RoboDK station: kr30 cnc template amana 46348 - paulina NEW THING.rdk

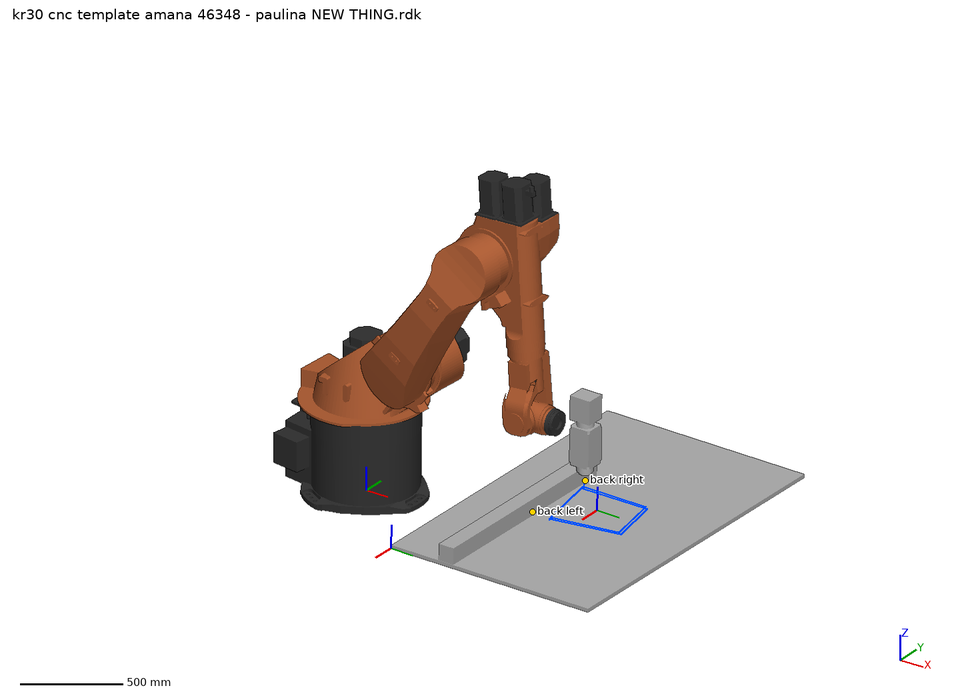
[picture v0: the station drawn from its stored meshes, robots at their saved joint values, targets as dots, program paths as lines]
Station kr30 cnc template amana 46348 - paulina NEW THING. Poses are relative to the parent item; angles as X-Y-Z fixed-axis rotations.
  - frame KUKA KR 30 HA Base at (0, 0, 0) mm
    - robot KUKA KR 30 HA: 6 axes, payload 30 kg, reach 2033 mm, repeatability 0.05 mm, weight 665 kg
        modified DH rows (alpha deg, a mm, theta deg, d mm): 0, 0, 0, 815; -90, 350, 0, 0; 0, 850, -90, 0; -90, 145, 0, 820; 90, 0, 0, 0; -90, 0, 180, 170
        joint limits [-185, -135, -120, -350, -119, -350] to [185, 35, 158, 350, 119, 350]; home [0, -90, 90, 0, 0, 0]; saved at [3.324, -56.878, 143.017, 183.529, 85.332, -180.023]
      - tool rc90 spindle mm, TCP at (267.95, 0.68, 160.99) mm, size 110 x 421.3 x 118 mm, geometry from rc90 spindle mm.stl
    - frame Tabletop at (921.82, -1104.91, 385) mm, rotated rx -0.93 ry -0.21 rz -89.9 deg
      - object tabletop CHECK HEIGHT at (-1839.9, 0, 0) mm, size 1839.9 x 1168.4 x 19 mm, geometry from kr30 tabletop mm.stl
      - object kr30 pipe jig base at (-1220, -610.6, 0) mm, size 1217.6 x 88.9 x 88.9 mm, geometry from kr30 pipe jig base.stl
      - frame Frame 3 at (-850, 630, 55.44) mm
      - target back right (Cartesian target) at (-1090.62, 392.95, 52.9) mm, rotated rx -9.38 ry 89.87 rz 80.74 deg; joints [0.828, -55.747, 144.821, 181.035, 88.274, -179.786] of KUKA KR 30 HA
      - target back left (Cartesian target) at (-646.79, 387.88, 55.43) mm, rotated rx -9.38 ry 89.87 rz 80.73 deg; joints [25.002, -54.059, 137.701, 205.384, 83.45, -182.49] of KUKA KR 30 HA
  - machining project Machining Settings: C:/Users/Research Office/Downloads/C1.apt | rotZ(0) | rotX(0)*rotY(0) | onStart | onPathStart | onApproach | onPoint | onRetract | onFinish | SetTool(%1) | onPathFinish
  - program Machining (400 instructions, listed below)
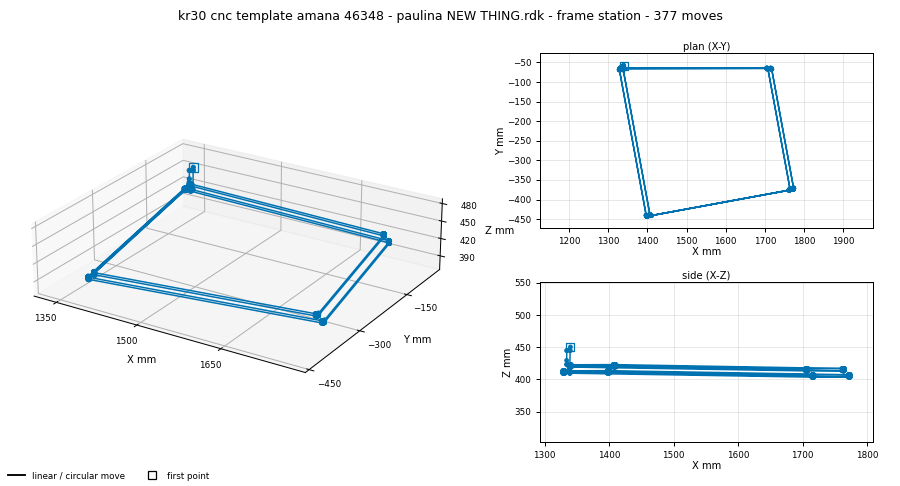
[picture p0: tool path of kr30 cnc template amana 46348 - paulina NEW THING.rdk in frame station, 377 of 377 moves have a stored position in this frame; points joined in program order, loops and branches not executed]

--- program Machining (robot KUKA KR 30 HA) ---
  Smooth(10)
  Print: /'1001'
  Print: /''
  Print: /'90 deg cut'
  Call SetTool(2)
  Set speed (100.0 mm/s)
  Set Ref.: Frame 3
  Set Tool: rc90 spindle mm
  Show rc90 spindle mm
  MoveJ 1 to (-195.95, -211.4, 20.67) mm, rotated rx -2.36 ry 89.88 rz 87.74 deg; joints [3.323, -57.284, 143.059, 183.53, 84.969, -180.046]
  MoveL 2 to (-192.49, -216.97, 15) mm, rotated rx 0 ry 90 rz 90.11 deg; joints [3.542, -56.953, 143.366, -176.241, 85.489, 179.974]
  MoveL 3 to (-192.49, -216.97, 15) mm, rotated rx 0 ry 90 rz 90.11 deg; joints [3.542, -56.953, 143.366, -176.241, 85.489, 179.974]
  Set speed (100.0 mm/s)
  MoveL 4 to (-192.49, -216.97, -0.32) mm, rotated rx 0 ry 90 rz 90.11 deg; joints [3.546, -55.577, 143.206, -176.242, 86.702, 180.054]
  Set speed (25.4 mm/s)
  MoveL 5 to (-192.49, -216.97, -6.37) mm, rotated rx 0 ry 90 rz 90.11 deg; joints [3.548, -55.032, 143.136, -176.242, 87.175, 180.085]
  MoveL 6 to (-192.02, -216.54, -7) mm, rotated rx 0 ry 90 rz 90.11 deg; joints [3.573, -54.966, 143.095, -176.217, 87.201, 180.086]
  Set speed (38.1 mm/s)
  MoveL 7 to (-187.83, -212.73, -7) mm, rotated rx 0 ry 90 rz 90.11 deg; joints [3.796, -54.884, 142.796, -175.994, 86.985, 180.063]
  MoveL 8 to (-187.84, -211.79, -7) mm, rotated rx 0 ry 90 rz 90.11 deg; joints [3.792, -54.864, 142.727, -175.997, 86.935, 180.06]
  Set speed (76.2 mm/s)
  MoveL 9 to (-188.01, -211.61, -7) mm, rotated rx 0 ry 90 rz 90.11 deg; joints [3.782, -54.861, 142.715, -176.007, 86.927, 180.06]
  MoveL 10 to (-188.15, -211.43, -7) mm, rotated rx 0 ry 90 rz 90.11 deg; joints [3.773, -54.857, 142.703, -176.016, 86.918, 180.06]
  MoveL 11 to (-188.32, -211.19, -7) mm, rotated rx 0 ry 90 rz 90.11 deg; joints [3.762, -54.852, 142.686, -176.027, 86.906, 180.059]
  MoveL 12 to (-188.46, -210.95, -7) mm, rotated rx 0 ry 90 rz 90.11 deg; joints [3.754, -54.848, 142.669, -176.035, 86.894, 180.059]
  MoveL 13 to (-188.57, -210.71, -7) mm, rotated rx 0 ry 90 rz 90.11 deg; joints [3.746, -54.843, 142.652, -176.042, 86.882, 180.058]
  MoveL 14 to (-188.66, -210.47, -7) mm, rotated rx 0 ry 90 rz 90.11 deg; joints [3.741, -54.838, 142.634, -176.048, 86.869, 180.057]
  MoveL 15 to (-188.72, -210.23, -7) mm, rotated rx 0 ry 90 rz 90.11 deg; joints [3.736, -54.833, 142.617, -176.053, 86.857, 180.057]
  MoveL 16 to (-188.77, -209.99, -7) mm, rotated rx 0 ry 90 rz 90.11 deg; joints [3.732, -54.828, 142.6, -176.056, 86.845, 180.056]
  MoveL 17 to (-188.8, -209.74, -7) mm, rotated rx 0 ry 90 rz 90.11 deg; joints [3.73, -54.823, 142.582, -176.059, 86.832, 180.055]
  MoveL 18 to (-188.81, -209.5, -7) mm, rotated rx 0 ry 90 rz 90.11 deg; joints [3.728, -54.818, 142.564, -176.06, 86.82, 180.054]
  MoveL 19 to (-188.81, 153.51, -7) mm, rotated rx 0 ry 90 rz 90.11 deg; joints [2.724, -44.301, 113.966, -176.857, 68.761, 179.117]
  MoveL 20 to (-188.81, 153.99, -7) mm, rotated rx 0 ry 90 rz 90.11 deg; joints [2.723, -44.283, 113.924, -176.858, 68.736, 179.116]
  MoveL 21 to (-188.8, 154.23, -7) mm, rotated rx 0 ry 90 rz 90.11 deg; joints [2.723, -44.275, 113.904, -176.858, 68.724, 179.116]
  MoveL 22 to (-188.76, 154.47, -7) mm, rotated rx 0 ry 90 rz 90.11 deg; joints [2.724, -44.266, 113.883, -176.856, 68.712, 179.115]
  MoveL 23 to (-188.71, 154.71, -7) mm, rotated rx 0 ry 90 rz 90.11 deg; joints [2.725, -44.257, 113.862, -176.854, 68.7, 179.113]
  MoveL 24 to (-188.64, 154.96, -7) mm, rotated rx 0 ry 90 rz 90.11 deg; joints [2.728, -44.248, 113.841, -176.851, 68.688, 179.112]
  MoveL 25 to (-188.55, 155.2, -7) mm, rotated rx 0 ry 90 rz 90.11 deg; joints [2.731, -44.24, 113.82, -176.848, 68.676, 179.11]
  MoveL 26 to (-188.43, 155.44, -7) mm, rotated rx 0 ry 90 rz 90.11 deg; joints [2.735, -44.231, 113.798, -176.843, 68.664, 179.107]
  MoveL 27 to (-188.35, 155.57, -7) mm, rotated rx 0 ry 90 rz 90.11 deg; joints [2.738, -44.226, 113.787, -176.839, 68.657, 179.106]
  MoveL 28 to (-188.27, 155.7, -7) mm, rotated rx 0 ry 90 rz 90.11 deg; joints [2.741, -44.221, 113.775, -176.836, 68.65, 179.104]
  MoveL 29 to (-188.18, 155.83, -7) mm, rotated rx 0 ry 90 rz 90.11 deg; joints [2.745, -44.216, 113.763, -176.832, 68.644, 179.103]
  MoveL 30 to (-188.08, 155.96, -7) mm, rotated rx 0 ry 90 rz 90.11 deg; joints [2.749, -44.211, 113.752, -176.827, 68.637, 179.101]
  MoveL 31 to (-187.95, 156.11, -7) mm, rotated rx 0 ry 90 rz 90.11 deg; joints [2.754, -44.206, 113.739, -176.822, 68.629, 179.098]
  MoveL 32 to (-187.8, 156.26, -7) mm, rotated rx 0 ry 90 rz 90.11 deg; joints [2.76, -44.2, 113.725, -176.815, 68.622, 179.096]
  MoveL 33 to (-187.66, 156.38, -7) mm, rotated rx 0 ry 90 rz 90.11 deg; joints [2.765, -44.195, 113.714, -176.809, 68.615, 179.093]
  MoveL 34 to (-187.52, 156.49, -7) mm, rotated rx 0 ry 90 rz 90.11 deg; joints [2.771, -44.191, 113.704, -176.803, 68.61, 179.091]
  MoveL 35 to (-187.28, 156.65, -7) mm, rotated rx 0 ry 90 rz 90.11 deg; joints [2.781, -44.185, 113.689, -176.793, 68.601, 179.087]
  MoveL 36 to (-187.04, 156.78, -7) mm, rotated rx 0 ry 90 rz 90.11 deg; joints [2.79, -44.18, 113.677, -176.782, 68.594, 179.082]
  MoveL 37 to (-186.8, 156.89, -7) mm, rotated rx 0 ry 90 rz 90.11 deg; joints [2.8, -44.176, 113.667, -176.772, 68.588, 179.078]
  MoveL 38 to (-186.55, 156.97, -7) mm, rotated rx 0 ry 90 rz 90.11 deg; joints [2.81, -44.172, 113.658, -176.761, 68.584, 179.074]
  MoveL 39 to (-186.31, 157.03, -7) mm, rotated rx 0 ry 90 rz 90.11 deg; joints [2.82, -44.17, 113.652, -176.75, 68.58, 179.071]
  MoveL 40 to (-186.07, 157.08, -7) mm, rotated rx 0 ry 90 rz 90.11 deg; joints [2.83, -44.168, 113.647, -176.74, 68.577, 179.067]
  MoveL 41 to (118.89, 212.92, -7) mm, rotated rx 0 ry 90 rz 90.11 deg; joints [14.55, -40.356, 104.549, -163.565, 64.177, 173.133]
  MoveL 42 to (119.13, 212.96, -7) mm, rotated rx 0 ry 90 rz 90.11 deg; joints [14.559, -40.353, 104.54, -163.555, 64.173, 173.127]
  MoveL 43 to (119.38, 212.98, -7) mm, rotated rx 0 ry 90 rz 90.11 deg; joints [14.568, -40.349, 104.532, -163.545, 64.17, 173.122]
  MoveL 44 to (119.62, 212.99, -7) mm, rotated rx 0 ry 90 rz 90.11 deg; joints [14.577, -40.347, 104.526, -163.534, 64.168, 173.117]
  MoveL 45 to (119.86, 212.97, -7) mm, rotated rx 0 ry 90 rz 90.11 deg; joints [14.586, -40.345, 104.522, -163.524, 64.167, 173.112]
  MoveL 46 to (120.1, 212.94, -7) mm, rotated rx 0 ry 90 rz 90.11 deg; joints [14.595, -40.344, 104.52, -163.513, 64.167, 173.107]
  MoveL 47 to (120.34, 212.88, -7) mm, rotated rx 0 ry 90 rz 90.11 deg; joints [14.605, -40.344, 104.519, -163.503, 64.167, 173.102]
  MoveL 48 to (120.58, 212.81, -7) mm, rotated rx 0 ry 90 rz 90.11 deg; joints [14.615, -40.344, 104.52, -163.492, 64.169, 173.098]
  MoveL 49 to (120.82, 212.71, -7) mm, rotated rx 0 ry 90 rz 90.11 deg; joints [14.625, -40.346, 104.523, -163.481, 64.172, 173.094]
  MoveL 50 to (121.07, 212.59, -7) mm, rotated rx 0 ry 90 rz 90.11 deg; joints [14.635, -40.348, 104.528, -163.471, 64.176, 173.09]
  MoveL 51 to (121.31, 212.44, -7) mm, rotated rx 0 ry 90 rz 90.11 deg; joints [14.645, -40.352, 104.535, -163.46, 64.181, 173.086]
  MoveL 52 to (121.55, 212.26, -7) mm, rotated rx 0 ry 90 rz 90.11 deg; joints [14.656, -40.356, 104.546, -163.448, 64.188, 173.083]
  MoveL 53 to (121.79, 212.04, -7) mm, rotated rx 0 ry 90 rz 90.11 deg; joints [14.667, -40.363, 104.56, -163.437, 64.197, 173.081]
  MoveL 54 to (121.93, 211.89, -7) mm, rotated rx 0 ry 90 rz 90.11 deg; joints [14.674, -40.367, 104.57, -163.431, 64.203, 173.079]
  MoveL 55 to (122.05, 211.74, -7) mm, rotated rx 0 ry 90 rz 90.11 deg; joints [14.68, -40.372, 104.581, -163.425, 64.209, 173.078]
  MoveL 56 to (122.16, 211.59, -7) mm, rotated rx 0 ry 90 rz 90.11 deg; joints [14.685, -40.377, 104.592, -163.42, 64.216, 173.078]
  MoveL 57 to (122.26, 211.43, -7) mm, rotated rx 0 ry 90 rz 90.11 deg; joints [14.691, -40.382, 104.603, -163.415, 64.223, 173.077]
  MoveL 58 to (122.39, 211.19, -7) mm, rotated rx 0 ry 90 rz 90.11 deg; joints [14.698, -40.39, 104.622, -163.408, 64.233, 173.077]
  MoveL 59 to (122.49, 210.95, -7) mm, rotated rx 0 ry 90 rz 90.11 deg; joints [14.704, -40.398, 104.641, -163.403, 64.244, 173.078]
  MoveL 60 to (122.57, 210.71, -7) mm, rotated rx 0 ry 90 rz 90.11 deg; joints [14.709, -40.407, 104.66, -163.398, 64.256, 173.079]
  MoveL 61 to (122.63, 210.47, -7) mm, rotated rx 0 ry 90 rz 90.11 deg; joints [14.714, -40.416, 104.68, -163.395, 64.267, 173.08]
  MoveL 62 to (122.81, 209.5, -7) mm, rotated rx 0 ry 90 rz 90.11 deg; joints [14.73, -40.452, 104.762, -163.383, 64.313, 173.087]
  MoveL 63 to (186.99, -140.96, -7) mm, rotated rx 0 ry 90 rz 90.11 deg; joints [22.176, -51.22, 131.007, -157.229, 79.633, 176.273]
  MoveL 64 to (187.07, -141.44, -7) mm, rotated rx 0 ry 90 rz 90.11 deg; joints [22.189, -51.232, 131.039, -157.218, 79.653, 176.279]
  MoveL 65 to (187.09, -141.68, -7) mm, rotated rx 0 ry 90 rz 90.11 deg; joints [22.194, -51.238, 131.056, -157.213, 79.663, 176.283]
  MoveL 66 to (187.09, -141.92, -7) mm, rotated rx 0 ry 90 rz 90.11 deg; joints [22.199, -51.245, 131.073, -157.209, 79.673, 176.286]
  MoveL 67 to (187.08, -142.16, -7) mm, rotated rx 0 ry 90 rz 90.11 deg; joints [22.203, -51.251, 131.091, -157.206, 79.684, 176.29]
  MoveL 68 to (187.04, -142.4, -7) mm, rotated rx 0 ry 90 rz 90.11 deg; joints [22.206, -51.258, 131.109, -157.204, 79.695, 176.294]
  MoveL 69 to (186.99, -142.65, -7) mm, rotated rx 0 ry 90 rz 90.11 deg; joints [22.208, -51.265, 131.128, -157.203, 79.706, 176.298]
  MoveL 70 to (186.91, -142.89, -7) mm, rotated rx 0 ry 90 rz 90.11 deg; joints [22.209, -51.272, 131.148, -157.202, 79.718, 176.303]
  MoveL 71 to (186.81, -143.13, -7) mm, rotated rx 0 ry 90 rz 90.11 deg; joints [22.209, -51.279, 131.168, -157.203, 79.729, 176.308]
  MoveL 72 to (186.69, -143.37, -7) mm, rotated rx 0 ry 90 rz 90.11 deg; joints [22.208, -51.287, 131.189, -157.205, 79.742, 176.314]
  MoveL 73 to (186.55, -143.61, -7) mm, rotated rx 0 ry 90 rz 90.11 deg; joints [22.206, -51.294, 131.21, -157.208, 79.754, 176.319]
  MoveL 74 to (186.36, -143.85, -7) mm, rotated rx 0 ry 90 rz 90.11 deg; joints [22.202, -51.303, 131.233, -157.213, 79.767, 176.326]
  MoveL 75 to (186.19, -144.05, -7) mm, rotated rx 0 ry 90 rz 90.11 deg; joints [22.197, -51.31, 131.252, -157.219, 79.779, 176.331]
  MoveL 76 to (185.98, -144.25, -7) mm, rotated rx 0 ry 90 rz 90.11 deg; joints [22.192, -51.317, 131.273, -157.225, 79.79, 176.337]
  MoveL 77 to (185.78, -144.4, -7) mm, rotated rx 0 ry 90 rz 90.11 deg; joints [22.186, -51.323, 131.289, -157.232, 79.8, 176.343]
  MoveL 78 to (185.59, -144.53, -7) mm, rotated rx 0 ry 90 rz 90.11 deg; joints [22.179, -51.328, 131.304, -157.239, 79.808, 176.347]
  MoveL 79 to (185.35, -144.66, -7) mm, rotated rx 0 ry 90 rz 90.11 deg; joints [22.171, -51.334, 131.321, -157.249, 79.817, 176.353]
  MoveL 80 to (185.1, -144.77, -7) mm, rotated rx 0 ry 90 rz 90.11 deg; joints [22.162, -51.339, 131.336, -157.259, 79.826, 176.358]
  MoveL 81 to (184.86, -144.86, -7) mm, rotated rx 0 ry 90 rz 90.11 deg; joints [22.152, -51.344, 131.349, -157.269, 79.833, 176.363]
  MoveL 82 to (184.62, -144.92, -7) mm, rotated rx 0 ry 90 rz 90.11 deg; joints [22.143, -51.348, 131.361, -157.279, 79.839, 176.368]
  MoveL 83 to (183.65, -145.1, -7) mm, rotated rx 0 ry 90 rz 90.11 deg; joints [22.102, -51.362, 131.402, -157.322, 79.861, 176.385]
  MoveL 84 to (-185.1, -212.63, -7) mm, rotated rx 0 ry 90 rz 90.11 deg; joints [3.949, -54.879, 142.775, -175.84, 86.969, 180.057]
  MoveL 85 to (-185.35, -212.66, -7) mm, rotated rx 0 ry 90 rz 90.11 deg; joints [3.936, -54.88, 142.778, -175.853, 86.972, 180.057]
  MoveL 86 to (-185.59, -212.67, -7) mm, rotated rx 0 ry 90 rz 90.11 deg; joints [3.922, -54.88, 142.781, -175.867, 86.973, 180.058]
  MoveL 87 to (-185.83, -212.67, -7) mm, rotated rx 0 ry 90 rz 90.11 deg; joints [3.908, -54.881, 142.781, -175.881, 86.974, 180.058]
  MoveL 88 to (-186.07, -212.64, -7) mm, rotated rx 0 ry 90 rz 90.11 deg; joints [3.895, -54.88, 142.781, -175.894, 86.974, 180.059]
  MoveL 89 to (-186.31, -212.6, -7) mm, rotated rx 0 ry 90 rz 90.11 deg; joints [3.881, -54.88, 142.779, -175.908, 86.972, 180.059]
  MoveL 90 to (-186.55, -212.54, -7) mm, rotated rx 0 ry 90 rz 90.11 deg; joints [3.867, -54.879, 142.776, -175.922, 86.97, 180.06]
  MoveL 91 to (-186.8, -212.45, -7) mm, rotated rx 0 ry 90 rz 90.11 deg; joints [3.853, -54.877, 142.771, -175.936, 86.966, 180.06]
  MoveL 92 to (-187.04, -212.35, -7) mm, rotated rx 0 ry 90 rz 90.11 deg; joints [3.839, -54.875, 142.764, -175.95, 86.962, 180.06]
  MoveL 93 to (-187.28, -212.21, -7) mm, rotated rx 0 ry 90 rz 90.11 deg; joints [3.825, -54.873, 142.756, -175.964, 86.956, 180.06]
  MoveL 94 to (-187.52, -212.05, -7) mm, rotated rx 0 ry 90 rz 90.11 deg; joints [3.811, -54.869, 142.745, -175.978, 86.948, 180.06]
  MoveL 95 to (-187.68, -211.93, -7) mm, rotated rx 0 ry 90 rz 90.11 deg; joints [3.801, -54.867, 142.737, -175.988, 86.942, 180.06]
  MoveL 96 to (-187.84, -211.79, -7) mm, rotated rx 0 ry 90 rz 90.11 deg; joints [3.792, -54.864, 142.727, -175.997, 86.935, 180.06]
  Set speed (38.1 mm/s)
  MoveL 97 to (-188.69, -212.73, -7) mm, rotated rx 0 ry 90 rz 90.11 deg; joints [3.748, -54.885, 142.8, -176.042, 86.988, 180.065]
  MoveL 98 to (-188.21, -213.16, -7) mm, rotated rx 0 ry 90 rz 90.11 deg; joints [3.776, -54.893, 142.829, -176.014, 87.009, 180.066]
  Set speed (25.4 mm/s)
  MoveL 99 to (-188.21, -213.16, -9.89) mm, rotated rx 0 ry 90 rz 90.11 deg; joints [3.777, -54.634, 142.794, -176.014, 87.232, 180.081]
  MoveL 100 to (-187.79, -212.68, -10.53) mm, rotated rx 0 ry 90 rz 90.11 deg; joints [3.799, -54.567, 142.75, -175.991, 87.254, 180.082]
  Set speed (38.1 mm/s)
  MoveL 101 to (-187.84, -211.79, -10.53) mm, rotated rx 0 ry 90 rz 90.11 deg; joints [3.793, -54.549, 142.684, -175.997, 87.207, 180.079]
  Set speed (76.2 mm/s)
  MoveL 102 to (-188.01, -211.61, -10.53) mm, rotated rx 0 ry 90 rz 90.11 deg; joints [3.783, -54.546, 142.672, -176.007, 87.198, 180.079]
  MoveL 103 to (-188.15, -211.43, -10.53) mm, rotated rx 0 ry 90 rz 90.11 deg; joints [3.774, -54.542, 142.66, -176.016, 87.19, 180.078]
  MoveL 104 to (-188.32, -211.19, -10.53) mm, rotated rx 0 ry 90 rz 90.11 deg; joints [3.763, -54.538, 142.643, -176.027, 87.178, 180.078]
  MoveL 105 to (-188.46, -210.95, -10.53) mm, rotated rx 0 ry 90 rz 90.11 deg; joints [3.755, -54.533, 142.626, -176.035, 87.165, 180.077]
  MoveL 106 to (-188.57, -210.71, -10.53) mm, rotated rx 0 ry 90 rz 90.11 deg; joints [3.747, -54.528, 142.609, -176.042, 87.153, 180.077]
  MoveL 107 to (-188.66, -210.47, -10.53) mm, rotated rx 0 ry 90 rz 90.11 deg; joints [3.742, -54.523, 142.592, -176.048, 87.141, 180.076]
  MoveL 108 to (-188.72, -210.23, -10.53) mm, rotated rx 0 ry 90 rz 90.11 deg; joints [3.737, -54.518, 142.574, -176.053, 87.128, 180.075]
  MoveL 109 to (-188.77, -209.99, -10.53) mm, rotated rx 0 ry 90 rz 90.11 deg; joints [3.733, -54.514, 142.557, -176.056, 87.116, 180.075]
  MoveL 110 to (-188.8, -209.74, -10.53) mm, rotated rx 0 ry 90 rz 90.11 deg; joints [3.731, -54.509, 142.539, -176.059, 87.103, 180.074]
  MoveL 111 to (-188.81, -209.5, -10.53) mm, rotated rx 0 ry 90 rz 90.11 deg; joints [3.729, -54.504, 142.522, -176.06, 87.09, 180.073]
  MoveL 112 to (-188.81, 153.51, -10.53) mm, rotated rx 0 ry 90 rz 90.11 deg; joints [2.724, -44.091, 113.934, -176.86, 68.937, 179.128]
  MoveL 113 to (-188.81, 153.99, -10.53) mm, rotated rx 0 ry 90 rz 90.11 deg; joints [2.723, -44.074, 113.892, -176.861, 68.913, 179.127]
  MoveL 114 to (-188.79, 154.23, -10.53) mm, rotated rx 0 ry 90 rz 90.11 deg; joints [2.723, -44.065, 113.871, -176.861, 68.901, 179.126]
  MoveL 115 to (-188.76, 154.47, -10.53) mm, rotated rx 0 ry 90 rz 90.11 deg; joints [2.724, -44.057, 113.85, -176.859, 68.889, 179.125]
  MoveL 116 to (-188.71, 154.71, -10.53) mm, rotated rx 0 ry 90 rz 90.11 deg; joints [2.726, -44.048, 113.829, -176.857, 68.877, 179.123]
  MoveL 117 to (-188.64, 154.96, -10.53) mm, rotated rx 0 ry 90 rz 90.11 deg; joints [2.728, -44.039, 113.808, -176.855, 68.865, 179.122]
  MoveL 118 to (-188.55, 155.2, -10.53) mm, rotated rx 0 ry 90 rz 90.11 deg; joints [2.732, -44.03, 113.787, -176.851, 68.852, 179.12]
  MoveL 119 to (-188.43, 155.44, -10.53) mm, rotated rx 0 ry 90 rz 90.11 deg; joints [2.736, -44.022, 113.766, -176.846, 68.84, 179.117]
  MoveL 120 to (-188.35, 155.57, -10.53) mm, rotated rx 0 ry 90 rz 90.11 deg; joints [2.739, -44.017, 113.754, -176.843, 68.833, 179.116]
  MoveL 121 to (-188.27, 155.7, -10.53) mm, rotated rx 0 ry 90 rz 90.11 deg; joints [2.742, -44.012, 113.743, -176.839, 68.827, 179.114]
  MoveL 122 to (-188.18, 155.83, -10.53) mm, rotated rx 0 ry 90 rz 90.11 deg; joints [2.746, -44.007, 113.731, -176.835, 68.82, 179.113]
  MoveL 123 to (-188.08, 155.96, -10.53) mm, rotated rx 0 ry 90 rz 90.11 deg; joints [2.75, -44.002, 113.719, -176.831, 68.813, 179.111]
  MoveL 124 to (-187.95, 156.11, -10.53) mm, rotated rx 0 ry 90 rz 90.11 deg; joints [2.755, -43.997, 113.706, -176.825, 68.806, 179.109]
  MoveL 125 to (-187.8, 156.26, -10.53) mm, rotated rx 0 ry 90 rz 90.11 deg; joints [2.761, -43.991, 113.693, -176.819, 68.798, 179.106]
  MoveL 126 to (-187.66, 156.38, -10.53) mm, rotated rx 0 ry 90 rz 90.11 deg; joints [2.766, -43.987, 113.682, -176.813, 68.792, 179.103]
  MoveL 127 to (-187.52, 156.49, -10.53) mm, rotated rx 0 ry 90 rz 90.11 deg; joints [2.772, -43.983, 113.672, -176.806, 68.786, 179.101]
  MoveL 128 to (-187.28, 156.65, -10.53) mm, rotated rx 0 ry 90 rz 90.11 deg; joints [2.781, -43.976, 113.657, -176.796, 68.777, 179.097]
  MoveL 129 to (-187.04, 156.78, -10.53) mm, rotated rx 0 ry 90 rz 90.11 deg; joints [2.791, -43.971, 113.645, -176.785, 68.77, 179.093]
  MoveL 130 to (-186.8, 156.89, -10.53) mm, rotated rx 0 ry 90 rz 90.11 deg; joints [2.801, -43.967, 113.634, -176.775, 68.764, 179.089]
  MoveL 131 to (-186.55, 156.97, -10.53) mm, rotated rx 0 ry 90 rz 90.11 deg; joints [2.811, -43.964, 113.626, -176.764, 68.76, 179.085]
  MoveL 132 to (-186.31, 157.03, -10.53) mm, rotated rx 0 ry 90 rz 90.11 deg; joints [2.82, -43.961, 113.62, -176.753, 68.756, 179.081]
  MoveL 133 to (-186.07, 157.08, -10.53) mm, rotated rx 0 ry 90 rz 90.11 deg; joints [2.83, -43.959, 113.615, -176.743, 68.753, 179.077]
  MoveL 134 to (118.89, 212.92, -10.53) mm, rotated rx 0 ry 90 rz 90.11 deg; joints [14.551, -40.165, 104.517, -163.586, 64.331, 173.183]
  MoveL 135 to (119.13, 212.96, -10.53) mm, rotated rx 0 ry 90 rz 90.11 deg; joints [14.56, -40.161, 104.508, -163.576, 64.327, 173.177]
  MoveL 136 to (119.38, 212.98, -10.53) mm, rotated rx 0 ry 90 rz 90.11 deg; joints [14.569, -40.158, 104.501, -163.565, 64.324, 173.172]
  MoveL 137 to (119.62, 212.99, -10.53) mm, rotated rx 0 ry 90 rz 90.11 deg; joints [14.578, -40.156, 104.495, -163.555, 64.322, 173.167]
  MoveL 138 to (119.86, 212.97, -10.53) mm, rotated rx 0 ry 90 rz 90.11 deg; joints [14.587, -40.154, 104.491, -163.545, 64.32, 173.162]
  MoveL 139 to (120.1, 212.94, -10.53) mm, rotated rx 0 ry 90 rz 90.11 deg; joints [14.596, -40.153, 104.488, -163.534, 64.32, 173.157]
  MoveL 140 to (120.34, 212.88, -10.53) mm, rotated rx 0 ry 90 rz 90.11 deg; joints [14.606, -40.153, 104.487, -163.524, 64.321, 173.152]
  MoveL 141 to (120.58, 212.81, -10.53) mm, rotated rx 0 ry 90 rz 90.11 deg; joints [14.616, -40.153, 104.488, -163.513, 64.322, 173.148]
  MoveL 142 to (120.83, 212.71, -10.53) mm, rotated rx 0 ry 90 rz 90.11 deg; joints [14.626, -40.155, 104.491, -163.502, 64.325, 173.144]
  MoveL 143 to (121.07, 212.59, -10.53) mm, rotated rx 0 ry 90 rz 90.11 deg; joints [14.636, -40.157, 104.497, -163.491, 64.329, 173.14]
  MoveL 144 to (121.31, 212.44, -10.53) mm, rotated rx 0 ry 90 rz 90.11 deg; joints [14.646, -40.16, 104.504, -163.48, 64.334, 173.136]
  MoveL 145 to (121.55, 212.26, -10.53) mm, rotated rx 0 ry 90 rz 90.11 deg; joints [14.657, -40.165, 104.515, -163.469, 64.341, 173.133]
  MoveL 146 to (121.79, 212.04, -10.53) mm, rotated rx 0 ry 90 rz 90.11 deg; joints [14.668, -40.171, 104.529, -163.458, 64.35, 173.131]
  MoveL 147 to (121.93, 211.89, -10.53) mm, rotated rx 0 ry 90 rz 90.11 deg; joints [14.675, -40.176, 104.539, -163.451, 64.357, 173.129]
  MoveL 148 to (122.05, 211.74, -10.53) mm, rotated rx 0 ry 90 rz 90.11 deg; joints [14.681, -40.18, 104.55, -163.446, 64.363, 173.129]
  MoveL 149 to (122.16, 211.59, -10.53) mm, rotated rx 0 ry 90 rz 90.11 deg; joints [14.687, -40.185, 104.561, -163.44, 64.369, 173.128]
  MoveL 150 to (122.26, 211.43, -10.53) mm, rotated rx 0 ry 90 rz 90.11 deg; joints [14.692, -40.19, 104.572, -163.436, 64.376, 173.128]
  MoveL 151 to (122.39, 211.19, -10.53) mm, rotated rx 0 ry 90 rz 90.11 deg; joints [14.699, -40.198, 104.59, -163.429, 64.387, 173.128]
  MoveL 152 to (122.49, 210.95, -10.53) mm, rotated rx 0 ry 90 rz 90.11 deg; joints [14.705, -40.207, 104.609, -163.424, 64.398, 173.128]
  MoveL 153 to (122.57, 210.71, -10.53) mm, rotated rx 0 ry 90 rz 90.11 deg; joints [14.71, -40.215, 104.629, -163.419, 64.409, 173.129]
  MoveL 154 to (122.63, 210.47, -10.53) mm, rotated rx 0 ry 90 rz 90.11 deg; joints [14.715, -40.224, 104.649, -163.416, 64.421, 173.13]
  MoveL 155 to (122.81, 209.5, -10.53) mm, rotated rx 0 ry 90 rz 90.11 deg; joints [14.731, -40.26, 104.731, -163.404, 64.467, 173.138]
  MoveL 156 to (186.99, -140.96, -10.53) mm, rotated rx 0 ry 90 rz 90.11 deg; joints [22.178, -50.961, 130.97, -157.243, 79.838, 176.361]
  MoveL 157 to (187.07, -141.44, -10.53) mm, rotated rx 0 ry 90 rz 90.11 deg; joints [22.191, -50.973, 131.003, -157.231, 79.858, 176.367]
  MoveL 158 to (187.09, -141.68, -10.53) mm, rotated rx 0 ry 90 rz 90.11 deg; joints [22.196, -50.979, 131.019, -157.227, 79.868, 176.37]
  MoveL 159 to (187.09, -141.92, -10.53) mm, rotated rx 0 ry 90 rz 90.11 deg; joints [22.201, -50.985, 131.037, -157.223, 79.879, 176.373]
  MoveL 160 to (187.08, -142.16, -10.53) mm, rotated rx 0 ry 90 rz 90.11 deg; joints [22.204, -50.992, 131.054, -157.22, 79.889, 176.377]
  MoveL 161 to (187.04, -142.4, -10.53) mm, rotated rx 0 ry 90 rz 90.11 deg; joints [22.207, -50.999, 131.073, -157.218, 79.9, 176.381]
  MoveL 162 to (186.99, -142.65, -10.53) mm, rotated rx 0 ry 90 rz 90.11 deg; joints [22.209, -51.005, 131.092, -157.217, 79.912, 176.386]
  MoveL 163 to (186.91, -142.89, -10.53) mm, rotated rx 0 ry 90 rz 90.11 deg; joints [22.21, -51.012, 131.111, -157.216, 79.923, 176.391]
  MoveL 164 to (186.81, -143.13, -10.53) mm, rotated rx 0 ry 90 rz 90.11 deg; joints [22.21, -51.02, 131.131, -157.217, 79.935, 176.396]
  MoveL 165 to (186.69, -143.37, -10.53) mm, rotated rx 0 ry 90 rz 90.11 deg; joints [22.209, -51.027, 131.152, -157.219, 79.948, 176.401]
  MoveL 166 to (186.54, -143.61, -10.53) mm, rotated rx 0 ry 90 rz 90.11 deg; joints [22.207, -51.035, 131.174, -157.222, 79.96, 176.407]
  MoveL 167 to (186.36, -143.85, -10.53) mm, rotated rx 0 ry 90 rz 90.11 deg; joints [22.204, -51.043, 131.197, -157.227, 79.973, 176.413]
  MoveL 168 to (186.19, -144.05, -10.53) mm, rotated rx 0 ry 90 rz 90.11 deg; joints [22.199, -51.05, 131.216, -157.232, 79.985, 176.419]
  MoveL 169 to (185.98, -144.25, -10.53) mm, rotated rx 0 ry 90 rz 90.11 deg; joints [22.193, -51.057, 131.236, -157.239, 79.996, 176.425]
  MoveL 170 to (185.78, -144.4, -10.53) mm, rotated rx 0 ry 90 rz 90.11 deg; joints [22.187, -51.063, 131.253, -157.246, 80.006, 176.43]
  MoveL 171 to (185.59, -144.53, -10.53) mm, rotated rx 0 ry 90 rz 90.11 deg; joints [22.181, -51.068, 131.268, -157.253, 80.014, 176.435]
  MoveL 172 to (185.35, -144.66, -10.53) mm, rotated rx 0 ry 90 rz 90.11 deg; joints [22.172, -51.074, 131.285, -157.262, 80.024, 176.441]
  MoveL 173 to (185.1, -144.77, -10.53) mm, rotated rx 0 ry 90 rz 90.11 deg; joints [22.163, -51.079, 131.299, -157.272, 80.032, 176.446]
  MoveL 174 to (184.86, -144.86, -10.53) mm, rotated rx 0 ry 90 rz 90.11 deg; joints [22.154, -51.084, 131.313, -157.282, 80.039, 176.451]
  MoveL 175 to (184.62, -144.92, -10.53) mm, rotated rx 0 ry 90 rz 90.11 deg; joints [22.144, -51.088, 131.324, -157.293, 80.046, 176.455]
  MoveL 176 to (183.65, -145.1, -10.53) mm, rotated rx 0 ry 90 rz 90.11 deg; joints [22.104, -51.102, 131.365, -157.336, 80.068, 176.472]
  MoveL 177 to (-185.1, -212.63, -10.53) mm, rotated rx 0 ry 90 rz 90.11 deg; joints [3.95, -54.564, 142.732, -175.84, 87.241, 180.076]
  MoveL 178 to (-185.35, -212.66, -10.53) mm, rotated rx 0 ry 90 rz 90.11 deg; joints [3.937, -54.565, 142.736, -175.853, 87.243, 180.077]
  MoveL 179 to (-185.59, -212.67, -10.53) mm, rotated rx 0 ry 90 rz 90.11 deg; joints [3.923, -54.565, 142.738, -175.867, 87.245, 180.077]
  MoveL 180 to (-185.83, -212.67, -10.53) mm, rotated rx 0 ry 90 rz 90.11 deg; joints [3.909, -54.565, 142.739, -175.881, 87.246, 180.078]
  MoveL 181 to (-186.07, -212.64, -10.53) mm, rotated rx 0 ry 90 rz 90.11 deg; joints [3.896, -54.565, 142.738, -175.894, 87.245, 180.078]
  MoveL 182 to (-186.31, -212.6, -10.53) mm, rotated rx 0 ry 90 rz 90.11 deg; joints [3.882, -54.564, 142.736, -175.908, 87.244, 180.079]
  MoveL 183 to (-186.55, -212.54, -10.53) mm, rotated rx 0 ry 90 rz 90.11 deg; joints [3.868, -54.563, 142.733, -175.922, 87.242, 180.079]
  MoveL 184 to (-186.8, -212.45, -10.53) mm, rotated rx 0 ry 90 rz 90.11 deg; joints [3.854, -54.562, 142.728, -175.936, 87.238, 180.079]
  MoveL 185 to (-187.04, -212.35, -10.53) mm, rotated rx 0 ry 90 rz 90.11 deg; joints [3.84, -54.56, 142.721, -175.95, 87.234, 180.079]
  MoveL 186 to (-187.28, -212.21, -10.53) mm, rotated rx 0 ry 90 rz 90.11 deg; joints [3.826, -54.557, 142.713, -175.964, 87.227, 180.079]
  MoveL 187 to (-187.52, -212.05, -10.53) mm, rotated rx 0 ry 90 rz 90.11 deg; joints [3.812, -54.554, 142.702, -175.978, 87.22, 180.079]
  MoveL 188 to (-187.68, -211.93, -10.53) mm, rotated rx 0 ry 90 rz 90.11 deg; joints [3.802, -54.552, 142.694, -175.988, 87.214, 180.079]
  MoveL 189 to (-187.84, -211.79, -10.53) mm, rotated rx 0 ry 90 rz 90.11 deg; joints [3.793, -54.549, 142.684, -175.997, 87.207, 180.079]
  Set speed (38.1 mm/s)
  MoveL 190 to (-188.73, -211.83, -10.53) mm, rotated rx 0 ry 90 rz 90.11 deg; joints [3.742, -54.551, 142.692, -176.048, 87.213, 180.081]
  MoveL 191 to (-188.97, -211.99, -10.53) mm, rotated rx 0 ry 90 rz 90.11 deg; joints [3.73, -54.555, 142.705, -176.06, 87.222, 180.082]
  MoveL 192 to (-190.08, -212.42, -10.53) mm, rotated rx 0 ry 90 rz 90.11 deg; joints [3.669, -54.564, 142.742, -176.122, 87.249, 180.086]
  Set speed (25.4 mm/s)
  MoveL 193 to (-190.08, -212.42, -15.89) mm, rotated rx 0 ry 90 rz 90.11 deg; joints [3.67, -54.084, 142.674, -176.121, 87.661, 180.114]
  MoveL 194 to (-189.44, -212.42, -16.53) mm, rotated rx 0 ry 90 rz 90.11 deg; joints [3.706, -54.027, 142.663, -176.085, 87.707, 180.116]
  Set speed (38.1 mm/s)
  MoveL 195 to (-188.81, -211.79, -16.53) mm, rotated rx 0 ry 90 rz 90.11 deg; joints [3.74, -54.014, 142.613, -176.052, 87.67, 180.113]
  Set speed (76.2 mm/s)
  MoveL 196 to (-188.81, 163.64, -16.53) mm, rotated rx 0 ry 90 rz 90.11 deg; joints [2.705, -43.372, 113.003, -176.877, 68.726, 179.122]
  MoveL 197 to (-188.8, 163.89, -16.53) mm, rotated rx 0 ry 90 rz 90.11 deg; joints [2.705, -43.363, 112.982, -176.877, 68.714, 179.122]
  MoveL 198 to (-188.77, 164.13, -16.53) mm, rotated rx 0 ry 90 rz 90.11 deg; joints [2.706, -43.355, 112.961, -176.876, 68.702, 179.121]
  MoveL 199 to (-188.72, 164.37, -16.53) mm, rotated rx 0 ry 90 rz 90.11 deg; joints [2.707, -43.346, 112.94, -176.874, 68.689, 179.119]
  MoveL 200 to (-188.65, 164.61, -16.53) mm, rotated rx 0 ry 90 rz 90.11 deg; joints [2.709, -43.337, 112.919, -176.871, 68.677, 179.118]
  MoveL 201 to (-188.56, 164.85, -16.53) mm, rotated rx 0 ry 90 rz 90.11 deg; joints [2.713, -43.328, 112.898, -176.867, 68.665, 179.116]
  MoveL 202 to (-188.44, 165.09, -16.53) mm, rotated rx 0 ry 90 rz 90.11 deg; joints [2.717, -43.319, 112.876, -176.862, 68.652, 179.114]
  MoveL 203 to (-188.37, 165.23, -16.53) mm, rotated rx 0 ry 90 rz 90.11 deg; joints [2.72, -43.314, 112.864, -176.859, 68.645, 179.112]
  MoveL 204 to (-188.29, 165.36, -16.53) mm, rotated rx 0 ry 90 rz 90.11 deg; joints [2.723, -43.31, 112.852, -176.856, 68.639, 179.111]
  MoveL 205 to (-188.19, 165.5, -16.53) mm, rotated rx 0 ry 90 rz 90.11 deg; joints [2.726, -43.305, 112.84, -176.852, 68.632, 179.109]
  MoveL 206 to (-188.09, 165.63, -16.53) mm, rotated rx 0 ry 90 rz 90.11 deg; joints [2.73, -43.3, 112.828, -176.847, 68.625, 179.107]
  MoveL 207 to (-187.96, 165.78, -16.53) mm, rotated rx 0 ry 90 rz 90.11 deg; joints [2.736, -43.294, 112.815, -176.841, 68.617, 179.104]
  MoveL 208 to (-187.8, 165.93, -16.53) mm, rotated rx 0 ry 90 rz 90.11 deg; joints [2.742, -43.288, 112.801, -176.835, 68.609, 179.102]
  MoveL 209 to (-187.66, 166.06, -16.53) mm, rotated rx 0 ry 90 rz 90.11 deg; joints [2.747, -43.283, 112.789, -176.829, 68.602, 179.099]
  MoveL 210 to (-187.52, 166.17, -16.53) mm, rotated rx 0 ry 90 rz 90.11 deg; joints [2.753, -43.279, 112.779, -176.823, 68.596, 179.097]
  MoveL 211 to (-187.28, 166.33, -16.53) mm, rotated rx 0 ry 90 rz 90.11 deg; joints [2.762, -43.273, 112.764, -176.812, 68.588, 179.093]
  MoveL 212 to (-187.04, 166.46, -16.53) mm, rotated rx 0 ry 90 rz 90.11 deg; joints [2.772, -43.268, 112.752, -176.802, 68.58, 179.089]
  MoveL 213 to (-186.8, 166.57, -16.53) mm, rotated rx 0 ry 90 rz 90.11 deg; joints [2.782, -43.264, 112.741, -176.791, 68.575, 179.085]
  MoveL 214 to (-186.55, 166.66, -16.53) mm, rotated rx 0 ry 90 rz 90.11 deg; joints [2.791, -43.26, 112.733, -176.78, 68.57, 179.081]
  MoveL 215 to (-186.31, 166.72, -16.53) mm, rotated rx 0 ry 90 rz 90.11 deg; joints [2.801, -43.258, 112.727, -176.77, 68.566, 179.077]
  MoveL 216 to (-186.07, 166.76, -16.53) mm, rotated rx 0 ry 90 rz 90.11 deg; joints [2.811, -43.256, 112.722, -176.759, 68.563, 179.073]
  MoveL 217 to (116.96, 222.25, -16.53) mm, rotated rx 0 ry 90 rz 90.11 deg; joints [14.391, -39.494, 103.67, -163.739, 64.143, 173.202]
  MoveL 218 to (117.44, 222.34, -16.53) mm, rotated rx 0 ry 90 rz 90.11 deg; joints [14.408, -39.486, 103.652, -163.719, 64.134, 173.191]
  MoveL 219 to (117.68, 222.35, -16.53) mm, rotated rx 0 ry 90 rz 90.11 deg; joints [14.417, -39.483, 103.644, -163.708, 64.132, 173.185]
  MoveL 220 to (117.93, 222.36, -16.53) mm, rotated rx 0 ry 90 rz 90.11 deg; joints [14.426, -39.48, 103.639, -163.698, 64.129, 173.18]
  MoveL 221 to (118.17, 222.34, -16.53) mm, rotated rx 0 ry 90 rz 90.11 deg; joints [14.435, -39.479, 103.635, -163.688, 64.128, 173.175]
  MoveL 222 to (118.41, 222.3, -16.53) mm, rotated rx 0 ry 90 rz 90.11 deg; joints [14.444, -39.478, 103.632, -163.677, 64.128, 173.171]
  MoveL 223 to (118.65, 222.24, -16.53) mm, rotated rx 0 ry 90 rz 90.11 deg; joints [14.454, -39.478, 103.632, -163.667, 64.129, 173.166]
  MoveL 224 to (118.89, 222.17, -16.53) mm, rotated rx 0 ry 90 rz 90.11 deg; joints [14.464, -39.478, 103.633, -163.656, 64.131, 173.162]
  MoveL 225 to (119.13, 222.07, -16.53) mm, rotated rx 0 ry 90 rz 90.11 deg; joints [14.473, -39.48, 103.636, -163.645, 64.134, 173.158]
  MoveL 226 to (119.38, 221.95, -16.53) mm, rotated rx 0 ry 90 rz 90.11 deg; joints [14.484, -39.482, 103.642, -163.634, 64.138, 173.154]
  MoveL 227 to (119.62, 221.79, -16.53) mm, rotated rx 0 ry 90 rz 90.11 deg; joints [14.494, -39.486, 103.65, -163.623, 64.143, 173.15]
  MoveL 228 to (119.86, 221.61, -16.53) mm, rotated rx 0 ry 90 rz 90.11 deg; joints [14.505, -39.491, 103.661, -163.612, 64.15, 173.147]
  MoveL 229 to (120, 221.49, -16.53) mm, rotated rx 0 ry 90 rz 90.11 deg; joints [14.511, -39.494, 103.668, -163.606, 64.155, 173.146]
  MoveL 230 to (120.13, 221.35, -16.53) mm, rotated rx 0 ry 90 rz 90.11 deg; joints [14.517, -39.498, 103.678, -163.6, 64.161, 173.144]
  MoveL 231 to (120.25, 221.22, -16.53) mm, rotated rx 0 ry 90 rz 90.11 deg; joints [14.523, -39.502, 103.687, -163.594, 64.167, 173.143]
  MoveL 232 to (120.35, 221.09, -16.53) mm, rotated rx 0 ry 90 rz 90.11 deg; joints [14.528, -39.506, 103.696, -163.589, 64.172, 173.143]
  MoveL 233 to (120.51, 220.85, -16.53) mm, rotated rx 0 ry 90 rz 90.11 deg; joints [14.537, -39.514, 103.714, -163.582, 64.183, 173.142]
  MoveL 234 to (120.65, 220.61, -16.53) mm, rotated rx 0 ry 90 rz 90.11 deg; joints [14.544, -39.522, 103.732, -163.575, 64.194, 173.142]
  MoveL 235 to (120.76, 220.36, -16.53) mm, rotated rx 0 ry 90 rz 90.11 deg; joints [14.55, -39.531, 103.751, -163.569, 64.205, 173.142]
  MoveL 236 to (120.84, 220.12, -16.53) mm, rotated rx 0 ry 90 rz 90.11 deg; joints [14.556, -39.539, 103.771, -163.565, 64.216, 173.143]
  MoveL 237 to (120.91, 219.88, -16.53) mm, rotated rx 0 ry 90 rz 90.11 deg; joints [14.561, -39.548, 103.791, -163.561, 64.228, 173.144]
  MoveL 238 to (120.96, 219.64, -16.53) mm, rotated rx 0 ry 90 rz 90.11 deg; joints [14.565, -39.557, 103.812, -163.558, 64.239, 173.146]
  MoveL 239 to (188.75, -150.61, -16.53) mm, rotated rx 0 ry 90 rz 90.11 deg; joints [22.442, -50.749, 131.545, -157.029, 80.581, 176.63]
  MoveL 240 to (188.79, -150.85, -16.53) mm, rotated rx 0 ry 90 rz 90.11 deg; joints [22.448, -50.754, 131.561, -157.023, 80.591, 176.633]
  MoveL 241 to (188.81, -151.09, -16.53) mm, rotated rx 0 ry 90 rz 90.11 deg; joints [22.453, -50.76, 131.578, -157.018, 80.601, 176.637]
  MoveL 242 to (188.81, -151.33, -16.53) mm, rotated rx 0 ry 90 rz 90.11 deg; joints [22.458, -50.766, 131.595, -157.014, 80.612, 176.64]
  MoveL 243 to (188.79, -151.58, -16.53) mm, rotated rx 0 ry 90 rz 90.11 deg; joints [22.462, -50.773, 131.613, -157.011, 80.623, 176.644]
  MoveL 244 to (188.75, -151.82, -16.53) mm, rotated rx 0 ry 90 rz 90.11 deg; joints [22.464, -50.779, 131.632, -157.009, 80.634, 176.649]
  MoveL 245 to (188.69, -152.06, -16.53) mm, rotated rx 0 ry 90 rz 90.11 deg; joints [22.466, -50.786, 131.65, -157.008, 80.645, 176.653]
  MoveL 246 to (188.61, -152.3, -16.53) mm, rotated rx 0 ry 90 rz 90.11 deg; joints [22.467, -50.793, 131.67, -157.008, 80.657, 176.658]
  MoveL 247 to (188.51, -152.54, -16.53) mm, rotated rx 0 ry 90 rz 90.11 deg; joints [22.467, -50.8, 131.69, -157.009, 80.669, 176.663]
  MoveL 248 to (188.38, -152.78, -16.53) mm, rotated rx 0 ry 90 rz 90.11 deg; joints [22.466, -50.807, 131.711, -157.011, 80.682, 176.669]
  MoveL 249 to (188.23, -153.02, -16.53) mm, rotated rx 0 ry 90 rz 90.11 deg; joints [22.464, -50.815, 131.733, -157.014, 80.695, 176.675]
  MoveL 250 to (188.04, -153.27, -16.53) mm, rotated rx 0 ry 90 rz 90.11 deg; joints [22.46, -50.822, 131.756, -157.019, 80.708, 176.681]
  MoveL 251 to (187.81, -153.51, -16.53) mm, rotated rx 0 ry 90 rz 90.11 deg; joints [22.454, -50.831, 131.78, -157.026, 80.722, 176.688]
  MoveL 252 to (187.67, -153.64, -16.53) mm, rotated rx 0 ry 90 rz 90.11 deg; joints [22.449, -50.835, 131.793, -157.031, 80.73, 176.693]
  MoveL 253 to (187.52, -153.75, -16.53) mm, rotated rx 0 ry 90 rz 90.11 deg; joints [22.445, -50.84, 131.806, -157.036, 80.737, 176.696]
  MoveL 254 to (187.28, -153.91, -16.53) mm, rotated rx 0 ry 90 rz 90.11 deg; joints [22.437, -50.846, 131.824, -157.045, 80.748, 176.702]
  MoveL 255 to (187.04, -154.05, -16.53) mm, rotated rx 0 ry 90 rz 90.11 deg; joints [22.428, -50.852, 131.841, -157.054, 80.758, 176.708]
  MoveL 256 to (186.8, -154.15, -16.53) mm, rotated rx 0 ry 90 rz 90.11 deg; joints [22.419, -50.857, 131.856, -157.064, 80.766, 176.713]
  MoveL 257 to (186.55, -154.24, -16.53) mm, rotated rx 0 ry 90 rz 90.11 deg; joints [22.41, -50.861, 131.869, -157.074, 80.773, 176.718]
  MoveL 258 to (186.31, -154.3, -16.53) mm, rotated rx 0 ry 90 rz 90.11 deg; joints [22.4, -50.865, 131.88, -157.085, 80.78, 176.722]
  MoveL 259 to (186.07, -154.34, -16.53) mm, rotated rx 0 ry 90 rz 90.11 deg; joints [22.39, -50.869, 131.891, -157.095, 80.786, 176.727]
  MoveL 260 to (-185.1, -222.31, -16.53) mm, rotated rx 0 ry 90 rz 90.11 deg; joints [3.991, -54.213, 143.363, -175.802, 88.22, 180.147]
  MoveL 261 to (-185.35, -222.34, -16.53) mm, rotated rx 0 ry 90 rz 90.11 deg; joints [3.977, -54.214, 143.366, -175.816, 88.222, 180.147]
  MoveL 262 to (-185.59, -222.36, -16.53) mm, rotated rx 0 ry 90 rz 90.11 deg; joints [3.963, -54.214, 143.369, -175.829, 88.224, 180.148]
  MoveL 263 to (-185.83, -222.35, -16.53) mm, rotated rx 0 ry 90 rz 90.11 deg; joints [3.95, -54.214, 143.369, -175.843, 88.225, 180.148]
  MoveL 264 to (-186.07, -222.33, -16.53) mm, rotated rx 0 ry 90 rz 90.11 deg; joints [3.936, -54.214, 143.369, -175.857, 88.225, 180.148]
  MoveL 265 to (-186.31, -222.28, -16.53) mm, rotated rx 0 ry 90 rz 90.11 deg; joints [3.922, -54.214, 143.367, -175.871, 88.223, 180.148]
  MoveL 266 to (-186.55, -222.22, -16.53) mm, rotated rx 0 ry 90 rz 90.11 deg; joints [3.908, -54.213, 143.364, -175.885, 88.221, 180.148]
  MoveL 267 to (-186.8, -222.14, -16.53) mm, rotated rx 0 ry 90 rz 90.11 deg; joints [3.894, -54.211, 143.359, -175.899, 88.217, 180.148]
  MoveL 268 to (-187.04, -222.03, -16.53) mm, rotated rx 0 ry 90 rz 90.11 deg; joints [3.879, -54.209, 143.352, -175.913, 88.212, 180.148]
  MoveL 269 to (-187.28, -221.9, -16.53) mm, rotated rx 0 ry 90 rz 90.11 deg; joints [3.865, -54.207, 143.344, -175.928, 88.206, 180.148]
  MoveL 270 to (-187.52, -221.74, -16.53) mm, rotated rx 0 ry 90 rz 90.11 deg; joints [3.851, -54.204, 143.333, -175.942, 88.199, 180.148]
  MoveL 271 to (-187.68, -221.61, -16.53) mm, rotated rx 0 ry 90 rz 90.11 deg; joints [3.841, -54.202, 143.324, -175.952, 88.192, 180.147]
  MoveL 272 to (-187.85, -221.46, -16.53) mm, rotated rx 0 ry 90 rz 90.11 deg; joints [3.831, -54.199, 143.315, -175.962, 88.185, 180.147]
  MoveL 273 to (-188.02, -221.27, -16.53) mm, rotated rx 0 ry 90 rz 90.11 deg; joints [3.82, -54.196, 143.302, -175.972, 88.176, 180.146]
  MoveL 274 to (-188.17, -221.09, -16.53) mm, rotated rx 0 ry 90 rz 90.11 deg; joints [3.811, -54.193, 143.289, -175.982, 88.166, 180.146]
  MoveL 275 to (-188.34, -220.85, -16.53) mm, rotated rx 0 ry 90 rz 90.11 deg; joints [3.801, -54.188, 143.272, -175.992, 88.154, 180.145]
  MoveL 276 to (-188.47, -220.61, -16.53) mm, rotated rx 0 ry 90 rz 90.11 deg; joints [3.792, -54.184, 143.255, -176, 88.142, 180.144]
  MoveL 277 to (-188.58, -220.36, -16.53) mm, rotated rx 0 ry 90 rz 90.11 deg; joints [3.785, -54.179, 143.238, -176.007, 88.129, 180.144]
  MoveL 278 to (-188.67, -220.12, -16.53) mm, rotated rx 0 ry 90 rz 90.11 deg; joints [3.779, -54.175, 143.221, -176.013, 88.116, 180.143]
  MoveL 279 to (-188.73, -219.88, -16.53) mm, rotated rx 0 ry 90 rz 90.11 deg; joints [3.775, -54.17, 143.204, -176.018, 88.104, 180.142]
  MoveL 280 to (-188.78, -219.64, -16.53) mm, rotated rx 0 ry 90 rz 90.11 deg; joints [3.771, -54.165, 143.186, -176.021, 88.091, 180.141]
  MoveL 281 to (-188.8, -219.4, -16.53) mm, rotated rx 0 ry 90 rz 90.11 deg; joints [3.769, -54.161, 143.169, -176.024, 88.078, 180.14]
  MoveL 282 to (-188.81, -219.16, -16.53) mm, rotated rx 0 ry 90 rz 90.11 deg; joints [3.768, -54.156, 143.151, -176.025, 88.065, 180.14]
  MoveL 283 to (-188.81, -211.79, -16.53) mm, rotated rx 0 ry 90 rz 90.11 deg; joints [3.74, -54.014, 142.613, -176.052, 87.67, 180.113]
  MoveL 284 to (-188.81, -211.79, -20.05) mm, rotated rx 0 ry 90 rz 90.11 deg; joints [3.741, -53.698, 142.567, -176.052, 87.939, 180.131]
  MoveL 285 to (-188.81, 163.64, -20.05) mm, rotated rx 0 ry 90 rz 90.11 deg; joints [2.705, -43.164, 112.968, -176.88, 68.899, 179.132]
  MoveL 286 to (-188.8, 163.89, -20.05) mm, rotated rx 0 ry 90 rz 90.11 deg; joints [2.705, -43.155, 112.947, -176.88, 68.887, 179.132]
  MoveL 287 to (-188.77, 164.13, -20.05) mm, rotated rx 0 ry 90 rz 90.11 deg; joints [2.706, -43.146, 112.926, -176.878, 68.875, 179.131]
  MoveL 288 to (-188.72, 164.37, -20.05) mm, rotated rx 0 ry 90 rz 90.11 deg; joints [2.708, -43.138, 112.905, -176.877, 68.863, 179.129]
  MoveL 289 to (-188.65, 164.61, -20.05) mm, rotated rx 0 ry 90 rz 90.11 deg; joints [2.71, -43.129, 112.884, -176.874, 68.85, 179.128]
  MoveL 290 to (-188.56, 164.85, -20.05) mm, rotated rx 0 ry 90 rz 90.11 deg; joints [2.713, -43.12, 112.863, -176.87, 68.838, 179.126]
  MoveL 291 to (-188.44, 165.09, -20.05) mm, rotated rx 0 ry 90 rz 90.11 deg; joints [2.718, -43.111, 112.841, -176.865, 68.825, 179.124]
  MoveL 292 to (-188.37, 165.23, -20.05) mm, rotated rx 0 ry 90 rz 90.11 deg; joints [2.72, -43.106, 112.829, -176.862, 68.818, 179.122]
  MoveL 293 to (-188.29, 165.36, -20.05) mm, rotated rx 0 ry 90 rz 90.11 deg; joints [2.724, -43.101, 112.817, -176.859, 68.811, 179.12]
  MoveL 294 to (-188.19, 165.5, -20.05) mm, rotated rx 0 ry 90 rz 90.11 deg; joints [2.727, -43.096, 112.805, -176.855, 68.804, 179.119]
  MoveL 295 to (-188.09, 165.63, -20.05) mm, rotated rx 0 ry 90 rz 90.11 deg; joints [2.731, -43.091, 112.793, -176.85, 68.797, 179.117]
  MoveL 296 to (-187.96, 165.78, -20.05) mm, rotated rx 0 ry 90 rz 90.11 deg; joints [2.736, -43.086, 112.78, -176.844, 68.79, 179.114]
  MoveL 297 to (-187.8, 165.93, -20.05) mm, rotated rx 0 ry 90 rz 90.11 deg; joints [2.742, -43.08, 112.766, -176.838, 68.782, 179.112]
  MoveL 298 to (-187.66, 166.06, -20.05) mm, rotated rx 0 ry 90 rz 90.11 deg; joints [2.748, -43.075, 112.754, -176.832, 68.775, 179.109]
  MoveL 299 to (-187.52, 166.17, -20.05) mm, rotated rx 0 ry 90 rz 90.11 deg; joints [2.753, -43.071, 112.744, -176.826, 68.769, 179.107]
  MoveL 300 to (-187.28, 166.33, -20.05) mm, rotated rx 0 ry 90 rz 90.11 deg; joints [2.763, -43.065, 112.729, -176.815, 68.76, 179.103]
  MoveL 301 to (-187.04, 166.46, -20.05) mm, rotated rx 0 ry 90 rz 90.11 deg; joints [2.773, -43.06, 112.717, -176.805, 68.753, 179.099]
  MoveL 302 to (-186.8, 166.57, -20.05) mm, rotated rx 0 ry 90 rz 90.11 deg; joints [2.782, -43.056, 112.706, -176.794, 68.747, 179.095]
  MoveL 303 to (-186.55, 166.66, -20.05) mm, rotated rx 0 ry 90 rz 90.11 deg; joints [2.792, -43.052, 112.698, -176.783, 68.743, 179.091]
  MoveL 304 to (-186.31, 166.72, -20.05) mm, rotated rx 0 ry 90 rz 90.11 deg; joints [2.802, -43.05, 112.692, -176.773, 68.739, 179.087]
  MoveL 305 to (-186.07, 166.76, -20.05) mm, rotated rx 0 ry 90 rz 90.11 deg; joints [2.812, -43.048, 112.687, -176.762, 68.736, 179.083]
  MoveL 306 to (116.96, 222.25, -20.05) mm, rotated rx 0 ry 90 rz 90.11 deg; joints [14.392, -39.302, 103.636, -163.759, 64.294, 173.251]
  MoveL 307 to (117.44, 222.34, -20.05) mm, rotated rx 0 ry 90 rz 90.11 deg; joints [14.409, -39.295, 103.617, -163.739, 64.285, 173.239]
  MoveL 308 to (117.68, 222.35, -20.05) mm, rotated rx 0 ry 90 rz 90.11 deg; joints [14.418, -39.292, 103.61, -163.728, 64.282, 173.234]
  MoveL 309 to (117.93, 222.36, -20.05) mm, rotated rx 0 ry 90 rz 90.11 deg; joints [14.427, -39.289, 103.604, -163.718, 64.28, 173.229]
  MoveL 310 to (118.17, 222.34, -20.05) mm, rotated rx 0 ry 90 rz 90.11 deg; joints [14.436, -39.288, 103.601, -163.708, 64.279, 173.224]
  MoveL 311 to (118.41, 222.3, -20.05) mm, rotated rx 0 ry 90 rz 90.11 deg; joints [14.445, -39.287, 103.598, -163.697, 64.279, 173.219]
  MoveL 312 to (118.65, 222.24, -20.05) mm, rotated rx 0 ry 90 rz 90.11 deg; joints [14.455, -39.286, 103.598, -163.687, 64.28, 173.215]
  MoveL 313 to (118.89, 222.17, -20.05) mm, rotated rx 0 ry 90 rz 90.11 deg; joints [14.465, -39.287, 103.599, -163.676, 64.281, 173.21]
  MoveL 314 to (119.13, 222.07, -20.05) mm, rotated rx 0 ry 90 rz 90.11 deg; joints [14.475, -39.289, 103.602, -163.665, 64.284, 173.206]
  MoveL 315 to (119.38, 221.95, -20.05) mm, rotated rx 0 ry 90 rz 90.11 deg; joints [14.485, -39.291, 103.608, -163.655, 64.288, 173.202]
  MoveL 316 to (119.62, 221.79, -20.05) mm, rotated rx 0 ry 90 rz 90.11 deg; joints [14.495, -39.295, 103.616, -163.644, 64.294, 173.199]
  MoveL 317 to (119.86, 221.61, -20.05) mm, rotated rx 0 ry 90 rz 90.11 deg; joints [14.506, -39.3, 103.627, -163.633, 64.301, 173.196]
  MoveL 318 to (120, 221.49, -20.05) mm, rotated rx 0 ry 90 rz 90.11 deg; joints [14.512, -39.303, 103.634, -163.626, 64.306, 173.194]
  MoveL 319 to (120.13, 221.35, -20.05) mm, rotated rx 0 ry 90 rz 90.11 deg; joints [14.519, -39.307, 103.644, -163.62, 64.312, 173.193]
  MoveL 320 to (120.25, 221.22, -20.05) mm, rotated rx 0 ry 90 rz 90.11 deg; joints [14.524, -39.311, 103.653, -163.615, 64.317, 173.192]
  MoveL 321 to (120.35, 221.09, -20.05) mm, rotated rx 0 ry 90 rz 90.11 deg; joints [14.529, -39.315, 103.662, -163.61, 64.323, 173.191]
  MoveL 322 to (120.51, 220.85, -20.05) mm, rotated rx 0 ry 90 rz 90.11 deg; joints [14.538, -39.323, 103.68, -163.602, 64.334, 173.191]
  MoveL 323 to (120.65, 220.61, -20.05) mm, rotated rx 0 ry 90 rz 90.11 deg; joints [14.545, -39.331, 103.698, -163.595, 64.345, 173.191]
  MoveL 324 to (120.76, 220.36, -20.05) mm, rotated rx 0 ry 90 rz 90.11 deg; joints [14.551, -39.339, 103.717, -163.59, 64.356, 173.191]
  MoveL 325 to (120.84, 220.12, -20.05) mm, rotated rx 0 ry 90 rz 90.11 deg; joints [14.557, -39.348, 103.737, -163.585, 64.367, 173.192]
  MoveL 326 to (120.91, 219.88, -20.05) mm, rotated rx 0 ry 90 rz 90.11 deg; joints [14.562, -39.357, 103.757, -163.581, 64.379, 173.193]
  MoveL 327 to (120.96, 219.64, -20.05) mm, rotated rx 0 ry 90 rz 90.11 deg; joints [14.566, -39.366, 103.778, -163.578, 64.39, 173.195]
  MoveL 328 to (188.75, -150.61, -20.05) mm, rotated rx 0 ry 90 rz 90.11 deg; joints [22.443, -50.487, 131.505, -157.041, 80.786, 176.718]
  MoveL 329 to (188.79, -150.85, -20.05) mm, rotated rx 0 ry 90 rz 90.11 deg; joints [22.45, -50.492, 131.522, -157.036, 80.796, 176.721]
  MoveL 330 to (188.81, -151.09, -20.05) mm, rotated rx 0 ry 90 rz 90.11 deg; joints [22.455, -50.498, 131.538, -157.031, 80.806, 176.724]
  MoveL 331 to (188.81, -151.33, -20.05) mm, rotated rx 0 ry 90 rz 90.11 deg; joints [22.46, -50.504, 131.556, -157.027, 80.817, 176.728]
  MoveL 332 to (188.79, -151.58, -20.05) mm, rotated rx 0 ry 90 rz 90.11 deg; joints [22.463, -50.51, 131.573, -157.024, 80.828, 176.732]
  MoveL 333 to (188.75, -151.82, -20.05) mm, rotated rx 0 ry 90 rz 90.11 deg; joints [22.466, -50.517, 131.592, -157.022, 80.839, 176.737]
  MoveL 334 to (188.69, -152.06, -20.05) mm, rotated rx 0 ry 90 rz 90.11 deg; joints [22.468, -50.523, 131.611, -157.021, 80.85, 176.741]
  MoveL 335 to (188.61, -152.3, -20.05) mm, rotated rx 0 ry 90 rz 90.11 deg; joints [22.469, -50.53, 131.63, -157.021, 80.862, 176.746]
  MoveL 336 to (188.51, -152.54, -20.05) mm, rotated rx 0 ry 90 rz 90.11 deg; joints [22.469, -50.537, 131.65, -157.021, 80.874, 176.751]
  MoveL 337 to (188.38, -152.78, -20.05) mm, rotated rx 0 ry 90 rz 90.11 deg; joints [22.468, -50.544, 131.671, -157.023, 80.887, 176.757]
  MoveL 338 to (188.23, -153.02, -20.05) mm, rotated rx 0 ry 90 rz 90.11 deg; joints [22.465, -50.552, 131.693, -157.027, 80.9, 176.763]
  MoveL 339 to (188.04, -153.27, -20.05) mm, rotated rx 0 ry 90 rz 90.11 deg; joints [22.461, -50.56, 131.716, -157.032, 80.913, 176.769]
  MoveL 340 to (187.81, -153.51, -20.05) mm, rotated rx 0 ry 90 rz 90.11 deg; joints [22.455, -50.568, 131.74, -157.039, 80.928, 176.776]
  MoveL 341 to (187.67, -153.64, -20.05) mm, rotated rx 0 ry 90 rz 90.11 deg; joints [22.451, -50.572, 131.753, -157.044, 80.936, 176.781]
  MoveL 342 to (187.52, -153.75, -20.05) mm, rotated rx 0 ry 90 rz 90.11 deg; joints [22.447, -50.577, 131.766, -157.049, 80.943, 176.784]
  MoveL 343 to (187.28, -153.91, -20.05) mm, rotated rx 0 ry 90 rz 90.11 deg; joints [22.439, -50.583, 131.784, -157.057, 80.954, 176.79]
  MoveL 344 to (187.04, -154.04, -20.05) mm, rotated rx 0 ry 90 rz 90.11 deg; joints [22.43, -50.589, 131.801, -157.067, 80.963, 176.796]
  MoveL 345 to (186.8, -154.15, -20.05) mm, rotated rx 0 ry 90 rz 90.11 deg; joints [22.421, -50.594, 131.816, -157.076, 80.972, 176.801]
  MoveL 346 to (186.55, -154.24, -20.05) mm, rotated rx 0 ry 90 rz 90.11 deg; joints [22.412, -50.598, 131.829, -157.087, 80.979, 176.806]
  MoveL 347 to (186.31, -154.3, -20.05) mm, rotated rx 0 ry 90 rz 90.11 deg; joints [22.402, -50.602, 131.84, -157.097, 80.986, 176.81]
  MoveL 348 to (186.07, -154.34, -20.05) mm, rotated rx 0 ry 90 rz 90.11 deg; joints [22.392, -50.605, 131.851, -157.108, 80.992, 176.815]
  MoveL 349 to (-185.1, -222.31, -20.05) mm, rotated rx 0 ry 90 rz 90.11 deg; joints [3.992, -53.893, 143.316, -175.802, 88.492, 180.167]
  MoveL 350 to (-185.35, -222.34, -20.05) mm, rotated rx 0 ry 90 rz 90.11 deg; joints [3.978, -53.894, 143.32, -175.815, 88.495, 180.167]
  MoveL 351 to (-185.59, -222.36, -20.05) mm, rotated rx 0 ry 90 rz 90.11 deg; joints [3.964, -53.894, 143.322, -175.829, 88.496, 180.168]
  MoveL 352 to (-185.83, -222.35, -20.05) mm, rotated rx 0 ry 90 rz 90.11 deg; joints [3.951, -53.894, 143.322, -175.843, 88.497, 180.168]
  MoveL 353 to (-186.07, -222.33, -20.05) mm, rotated rx 0 ry 90 rz 90.11 deg; joints [3.937, -53.894, 143.322, -175.857, 88.497, 180.168]
  MoveL 354 to (-186.31, -222.28, -20.05) mm, rotated rx 0 ry 90 rz 90.11 deg; joints [3.923, -53.894, 143.32, -175.871, 88.495, 180.168]
  MoveL 355 to (-186.55, -222.22, -20.05) mm, rotated rx 0 ry 90 rz 90.11 deg; joints [3.909, -53.893, 143.317, -175.885, 88.493, 180.168]
  MoveL 356 to (-186.8, -222.14, -20.05) mm, rotated rx 0 ry 90 rz 90.11 deg; joints [3.895, -53.891, 143.312, -175.899, 88.489, 180.168]
  MoveL 357 to (-187.04, -222.03, -20.05) mm, rotated rx 0 ry 90 rz 90.11 deg; joints [3.88, -53.89, 143.305, -175.913, 88.485, 180.168]
  MoveL 358 to (-187.28, -221.9, -20.05) mm, rotated rx 0 ry 90 rz 90.11 deg; joints [3.866, -53.887, 143.297, -175.927, 88.479, 180.167]
  MoveL 359 to (-187.52, -221.74, -20.05) mm, rotated rx 0 ry 90 rz 90.11 deg; joints [3.852, -53.885, 143.286, -175.942, 88.471, 180.167]
  MoveL 360 to (-187.68, -221.61, -20.05) mm, rotated rx 0 ry 90 rz 90.11 deg; joints [3.842, -53.882, 143.278, -175.951, 88.464, 180.166]
  MoveL 361 to (-187.85, -221.46, -20.05) mm, rotated rx 0 ry 90 rz 90.11 deg; joints [3.832, -53.88, 143.268, -175.961, 88.457, 180.166]
  MoveL 362 to (-188.02, -221.27, -20.05) mm, rotated rx 0 ry 90 rz 90.11 deg; joints [3.821, -53.876, 143.255, -175.972, 88.448, 180.166]
  MoveL 363 to (-188.17, -221.09, -20.05) mm, rotated rx 0 ry 90 rz 90.11 deg; joints [3.812, -53.873, 143.242, -175.981, 88.438, 180.165]
  MoveL 364 to (-188.34, -220.85, -20.05) mm, rotated rx 0 ry 90 rz 90.11 deg; joints [3.802, -53.869, 143.226, -175.991, 88.426, 180.164]
  MoveL 365 to (-188.47, -220.61, -20.05) mm, rotated rx 0 ry 90 rz 90.11 deg; joints [3.793, -53.864, 143.209, -176, 88.413, 180.163]
  MoveL 366 to (-188.58, -220.36, -20.05) mm, rotated rx 0 ry 90 rz 90.11 deg; joints [3.786, -53.86, 143.192, -176.007, 88.401, 180.163]
  MoveL 367 to (-188.67, -220.12, -20.05) mm, rotated rx 0 ry 90 rz 90.11 deg; joints [3.78, -53.856, 143.174, -176.013, 88.388, 180.162]
  MoveL 368 to (-188.73, -219.88, -20.05) mm, rotated rx 0 ry 90 rz 90.11 deg; joints [3.776, -53.851, 143.157, -176.017, 88.375, 180.161]
  MoveL 369 to (-188.78, -219.64, -20.05) mm, rotated rx 0 ry 90 rz 90.11 deg; joints [3.772, -53.847, 143.14, -176.021, 88.362, 180.16]
  MoveL 370 to (-188.8, -219.4, -20.05) mm, rotated rx 0 ry 90 rz 90.11 deg; joints [3.77, -53.842, 143.122, -176.023, 88.349, 180.159]
  MoveL 371 to (-188.81, -219.16, -20.05) mm, rotated rx 0 ry 90 rz 90.11 deg; joints [3.769, -53.838, 143.105, -176.025, 88.336, 180.158]
  MoveL 372 to (-188.81, -211.79, -20.05) mm, rotated rx 0 ry 90 rz 90.11 deg; joints [3.741, -53.698, 142.567, -176.052, 87.939, 180.131]
  Set speed (38.1 mm/s)
  MoveL 373 to (-189.51, -211.15, -20.05) mm, rotated rx 0 ry 90 rz 90.11 deg; joints [3.699, -53.687, 142.524, -176.093, 87.907, 180.13]
  MoveL 374 to (-195.54, -211.76, -20.05) mm, rotated rx 0 ry 90 rz 90.11 deg; joints [3.361, -53.703, 142.595, -176.431, 87.962, 180.14]
  MoveL 375 to (-196.17, -211.82, -19.42) mm, rotated rx 0 ry 90 rz 90.11 deg; joints [3.326, -53.762, 142.611, -176.467, 87.919, 180.138]
  Set speed (100.0 mm/s)
  MoveL 376 to (-196.17, -211.82, 15) mm, rotated rx 0 ry 90 rz 90.11 deg; joints [3.316, -56.836, 143.004, -176.466, 85.243, 179.973]
  MoveL 377 to (-196.17, -211.82, 15) mm, rotated rx 0 ry 90 rz 90.11 deg; joints [3.316, -56.836, 143.004, -176.466, 85.243, 179.973]
